// TIA Portal V17 export
// export: Created 2025-06-26T06:33:59.0377873Z, ExportSetting WithDefaults, DisplayName Totally Integrated Automation Portal, DisplayVersion V17 Update 8, DisplayName TIA Portal Openness, DisplayVersion V17 Update 8, DisplayName TIA Portal Version Control Interface, DisplayVersion V17, DisplayName STEP 7 Professional, DisplayVersion V17 Update 8, DisplayName STEP 7 Safety, DisplayVersion V17 Update 6, DisplayName WinCC Advanced, DisplayVersion V17 Update 8
DATA_BLOCK "DB_Heatbooster"   // DB19
{ S7_Optimized_Access := 'TRUE' }
VERSION : 0.1
// stored: AutoNumber true, DBAccessibleFromOPCUA true, IsOnlyStoredInLoadMemory false, IsRetainMemResEnabled false, IsWriteProtectedInAS false, MemoryReserve 0
   VAR
      AI : Struct
         HBL_TT_502 { S7_SetPoint := 'True'} : "stCalcValue";   // Compressor discharge popoff temperature
         HBL_PT_503 { S7_SetPoint := 'True'} : "stCalcValue";   // Compressor discharge pressure
         HBL_TT_504 { S7_SetPoint := 'True'} : "stCalcValue";   // Compressor discharge temperature
         HBL_LT_510 { S7_SetPoint := 'True'} : "stCalcValue";   // Steam generator condensate level
         HBL_PT_511 { S7_SetPoint := 'True'} : "stCalcValue";   // Heat sink discharge pressure
         HBL_TT_512 { S7_SetPoint := 'True'} : "stCalcValue";   // Heat sink discharge temperature
         HBL_TT_516 { S7_SetPoint := 'True'} : "stCalcValue";   // Steam generator suction temperature
         HBL_PT_517 { S7_SetPoint := 'True'} : "stCalcValue";   // Steam generator suction pressure
         HBL_TT_518 { S7_SetPoint := 'True'} : "stCalcValue";   // Heat sink discharge process temperature
         HBL_PT_519 { S7_SetPoint := 'True'} : "stCalcValue";   // Heat sink discharge process pressure
         HBL_FT_520 { S7_SetPoint := 'True'} : "stCalcValue";   // Refrigerant flow
         HBL_TT_530 { S7_SetPoint := 'True'} : "stCalcValue";   // Expansion valve B discharge temperature
         HBL_PT_531 { S7_SetPoint := 'True'} : "stCalcValue";   // Expansion valve B discharge pressure
         HBL_TT_532 { S7_SetPoint := 'True'} : "stCalcValue";   // Heat source discharge B temperature
         HBL_TT_533 { S7_SetPoint := 'True'} : "stCalcValue";   // Evaporator B discharge temperature
         HBL_PT_534 { S7_SetPoint := 'True'} : "stCalcValue";   // Evaporator B discharge pressure
         HBL_AT_535 { S7_SetPoint := 'True'} : "stCalcValue";   // Evaporator B steam quality
         HBL_TT_540 { S7_SetPoint := 'True'} : "stCalcValue";   // Expansion valve A discharge temperature
         HBL_PT_541 { S7_SetPoint := 'True'} : "stCalcValue";   // Expansion valve A discharge pressure
         HBL_TT_542 { S7_SetPoint := 'True'} : "stCalcValue";   // Heat source discharge temperature
         HBL_TT_543 { S7_SetPoint := 'True'} : "stCalcValue";   // Evaporator A discharge temperature
         HBL_PT_544 { S7_SetPoint := 'True'} : "stCalcValue";   // Evaporator A discharge pressure
         HBL_AT_545 { S7_SetPoint := 'True'} : "stCalcValue";   // Evaporator A steam quality
         HBL_TT_546 { S7_SetPoint := 'True'} : "stCalcValue";   // Heat source suction temperature
         HBL_PT_547 { S7_SetPoint := 'True'} : "stCalcValue";   // Heast source suction pressure
         HBL_TT_571 { S7_SetPoint := 'True'} : "stCalcValue";   // Compressor suction temperature
         HBL_PT_572 { S7_SetPoint := 'True'} : "stCalcValue";   // Compressor suction pressure
         HBL_TT_573 { S7_SetPoint := 'True'} : "stCalcValue";   // Expansion valve suction temperature
         HBL_LT_610 { S7_SetPoint := 'True'} : "stCalcValue";   // HP receiver refrigerant level
         HBL_TT_611 { S7_SetPoint := 'True'} : "stCalcValue";   // Steam generator discharge temperature
         HBL_PT_612 { S7_SetPoint := 'True'} : "stCalcValue";   // Steam generator discharge pressure
         HBL_CT_615 { S7_SetPoint := 'True'} : "stCalcValue";   // Gas detector PSV discharge pipe
         HBL_PT_618 { S7_SetPoint := 'True'} : "stCalcValue";   // HP Receiver pressure
         HBL_PT_635 { S7_SetPoint := 'True'} : "stCalcValue";   // Oil separator stage 1 oil return pressure
         HBL_PT_636 { S7_SetPoint := 'True'} : "stCalcValue";   // Oil separator stage 2 oil return pressure
         HBL_LT_650 { S7_SetPoint := 'True'} : "stCalcValue";   // Heat source condensate buffer tank level
         HBL_PT_651 { S7_SetPoint := 'True'} : "stCalcValue";   // Heat source condensate buffer tank pressure
         HBL_PT_701 { S7_SetPoint := 'True'} : "stCalcValue";   // Filter dryer suction pressure
         HBL_PT_702 { S7_SetPoint := 'True'} : "stCalcValue";   // Filter dryer discharge pressure
         HBL_PT_703 { S7_SetPoint := 'True'} : "stCalcValue";   // Filter dryer differential pressure
         CPC_LT_870 { S7_SetPoint := 'True'} : "stCalcValue";   // CPC tank refrigerant level
         CPC_TT_871 { S7_SetPoint := 'True'} : "stCalcValue";   // CPC tank refrigerant temperature
         CPC_PT_872 { S7_SetPoint := 'True'} : "stCalcValue";   // CPC tank refrigerant pressure
         CPC_PT_862 { S7_SetPoint := 'True'} : "stCalcValue";   // CPC pump discharge pressure
         HBL_TT_901 { S7_SetPoint := 'True'} : "stCalcValue";   // Heat sink suction temperature
         HBL_PT_902 { S7_SetPoint := 'True'} : "stCalcValue";   // Heat sink suction pressure
         HBL_TT_03 { S7_SetPoint := 'True'} : "stCalcValue";   // Oil sump oil temperature
         HBL_TT_16 { S7_SetPoint := 'True'} : "stCalcValue";   // Container air temperature
         HBL_TT_17 { S7_SetPoint := 'True'} : "stCalcValue";   // Control cabinet air temperature
         HBL_TT_18 { S7_SetPoint := 'True'} : "stCalcValue";   // Ambient air temperature
         HBL_TT_20 { S7_SetPoint := 'True'} : "stCalcValue";   // Compressor motor winding temperature
         HBL_TT_21 { S7_SetPoint := 'True'} : "stCalcValue";   // Oil sump wall temperature left
         HBL_TT_22 { S7_SetPoint := 'True'} : "stCalcValue";   // Oil sump wall temperature right
         HBL_TT_23 { S7_SetPoint := 'True'} : "stCalcValue";   // Compressor motor U-winding temperature
         HBL_TT_24 { S7_SetPoint := 'True'} : "stCalcValue";   // Compressor motor V-winding temperature
         HBL_TT_25 { S7_SetPoint := 'True'} : "stCalcValue";   // Compressor motor W-winding temperature
         HBL_TT_26 { S7_SetPoint := 'True'} : "stCalcValue";   // Compressor motor D bearing temperature
         HBL_TT_27 { S7_SetPoint := 'True'} : "stCalcValue";   // Compressor motor N bearing temperature
         HBL_PT_05 { S7_SetPoint := 'True'} : "stCalcValue";   // Crankcase gas pressure
         HBL_PT_06 { S7_SetPoint := 'True'} : "stCalcValue";   // Oil pump discharge pressure
         HBL_PT_17 { S7_SetPoint := 'True'} : "stCalcValue";   // Oil gallery pressure
         HBL_CT_01 { S7_SetPoint := 'True'} : "stCalcValue";   // Gas detector Heatbooster (optional)
         HBL_CT_03 { S7_SetPoint := 'True'} : "stCalcValue";   // Gas detector container (optional)
         SSC_TT_01 { S7_SetPoint := 'True'} : "stCalcValue";   // SSC seal suction temperature
         SSC_TT_02 { S7_SetPoint := 'True'} : "stCalcValue";   // SSC seal discharge temperature
         SSC_TT_03 { S7_SetPoint := 'True'} : "stCalcValue";   // SSC barrier fluid circulation pump suction temperature
         SSC_TT_04 { S7_SetPoint := 'True'} : "stCalcValue";   // SSC barrier fluid heat exchanger temperature
         SSC_PIT_01 { S7_SetPoint := 'True'} : "stCalcValue";   // SSC barrier fluid accumulator pressure
         SSC_PDT_01 { S7_SetPoint := 'True'} : "stCalcValue";   // SSC barrier fluid circulation pump differential pressure
         SSC_LT_01 { S7_SetPoint := 'True'} : "stCalcValue";   // SSC barrier fluid reservoir level
         HBL_VT_01 { S7_SetPoint := 'True'} : "stCalcValue";   // [?] Oil sump oil viscosity
         HBL_TT_36 { S7_SetPoint := 'True'} : "stCalcValue";   // [C] Oil sump oil viscosity probe temperature
      END_STRUCT;
      Calc : Struct
         Compressor : Struct
            CrankcaseSaturationTemperature { S7_SetPoint := 'True'} : "stCalcValue";   // C
            CrankcaseSuperheat { S7_SetPoint := 'True'} : "stCalcValue";   // C
            VolumetricEfficiency { S7_SetPoint := 'True'} : "stCalcValue";   // %
            IsentropicEfficiency { S7_SetPoint := 'True'} : "stCalcValue";   // %
            Massflow { S7_SetPoint := 'True'} : "stCalcValue";   // kg/h
         END_STRUCT;
         HeatSink : Struct
            DeltaT { S7_SetPoint := 'True'} : "stCalcValue";
            Pinch { S7_SetPoint := 'True'} : "stCalcValue";
            HeatRate { S7_SetPoint := 'True'} : "stCalcValue";
            DeltaP { S7_SetPoint := 'True'} : "stCalcValue";
            Massflow { S7_SetPoint := 'True'} : "stCalcValue";
         END_STRUCT;
         HeatSource : Struct
            DeltaT { S7_SetPoint := 'True'} : "stCalcValue";
            Pinch { S7_SetPoint := 'True'} : "stCalcValue";
            HeatRate { S7_SetPoint := 'True'} : "stCalcValue";
            DeltaP { S7_SetPoint := 'True'} : "stCalcValue";
            TemperatureRateOfChange { S7_SetPoint := 'True'} : "stCalcValue";
            Massflow { S7_SetPoint := 'True'} : "stCalcValue";
         END_STRUCT;
         HighPressPart : Struct
            CompressorSaturationTemperature { S7_SetPoint := 'True'} : "stCalcValue";
            CompressorSuperheat { S7_SetPoint := 'True'} : "stCalcValue";
            CondenserSaturationTemperature { S7_SetPoint := 'True'} : "stCalcValue";
            CondenserSubcooling { S7_SetPoint := 'True'} : "stCalcValue";
            ExpansionValveSubcooling { S7_SetPoint := 'True'} : "stCalcValue";
            CondenserDeltaP { S7_SetPoint := 'True'} : "stCalcValue";
         END_STRUCT;
         LowPressPart : Struct
            EvaporatorSuperheat { S7_SetPoint := 'True'} : "stCalcValue";
            CompressorSuperheat { S7_SetPoint := 'True'} : "stCalcValue";
            EvaporatorSaturationTemperature { S7_SetPoint := 'True'} : "stCalcValue";
            CompressorSaturationTemperature { S7_SetPoint := 'True'} : "stCalcValue";
         END_STRUCT;
         System : Struct
            Quality { S7_SetPoint := 'True'} : "stCalcValue";
            COP { S7_SetPoint := 'True'} : "stCalcValue";
            ElectricalPower { S7_SetPoint := 'True'} : "stCalcValue";
            TemperatureLift { S7_SetPoint := 'True'} : "stCalcValue";
            MotorEfficiency { S7_SetPoint := 'True'} : "stCalcValue";
            FMEP { S7_SetPoint := 'True'} : "stCalcValue";
         END_STRUCT;
         Auxiliary : Struct
            ShaftSealDeltaT { S7_SetPoint := 'True'} : "stCalcValue";
            CPCPumpDeltaP { S7_SetPoint := 'True'} : "stCalcValue";
         END_STRUCT;
         Misc : Struct
            EvaporatorDischargePressureMean { S7_SetPoint := 'True'} : "stCalcValue";
            EvaporatorDischargeTemperatureMin { S7_SetPoint := 'True'} : "stCalcValue";
            EvaporatorDischargeTemperatureMean { S7_SetPoint := 'True'} : "stCalcValue";
            OilFilterDeltaP { S7_SetPoint := 'True'} : "stCalcValue";
         END_STRUCT;
      END_STRUCT;
      DI : Struct
         HBL_FS_01 : Bool;
         HBL_FS_02 : Bool;
         HBL_LS_632 : Bool;
         HBL_LS_633 : Bool;
         CPC_LS_864 : Bool;
         VPNUserConnected : Bool;
      END_STRUCT;
      "DO" : Struct
         HBL_EC_01 : Bool;
         HBL_EC_02 : Bool;
         HBL_HV_630 : Bool;
         HBL_HV_114 : Bool;
         HBL_HV_115 : Bool;
         HBL_HV_860 : Bool;
         HBL_HV_861 : Bool;
         SSC_P_01 : Bool;
         SSC_F_01 : Bool;
         SSC_P_02 : Bool;
         CPC_P_01 : Bool;
         SpareContactor1 : Bool;
         SpareContactor2 : Bool;
         HBL_HV_631 : Bool;
      END_STRUCT;
      Inverter : Struct
         HBL_SC_01_A1 { S7_SetPoint := 'True'} : "stCalcValue";   // Container ventilation fan speed
         HBL_SC_01_A2 { S7_SetPoint := 'True'} : "stCalcValue";   // Container ventilation fan torque
         HBL_SC_01_A3 { S7_SetPoint := 'True'} : "stCalcValue";   // Container ventilation fan power
         HBL_SC_02_A1 { S7_SetPoint := 'True'} : "stCalcValue";   // Compressor lubrication pump speed
         HBL_SC_02_A2 { S7_SetPoint := 'True'} : "stCalcValue";   // Compressor lubrication pump torque
         HBL_SC_02_A3 { S7_SetPoint := 'True'} : "stCalcValue";   // Compressor lubrication pump power
         HBL_SC_03_A1 { S7_SetPoint := 'True'} : "stCalcValue";   // CPC pump speed
         HBL_SC_03_A2 { S7_SetPoint := 'True'} : "stCalcValue";   // CPC pump torque
         HBL_SC_03_A3 { S7_SetPoint := 'True'} : "stCalcValue";   // CPC pump power
         HBL_SC_10_A1 { S7_SetPoint := 'True'} : "stCalcValue";   // Compressor motor speed
         HBL_SC_10_A2 { S7_SetPoint := 'True'} : "stCalcValue";   // Compressor motor torque
         HBL_SC_10_A3 { S7_SetPoint := 'True'} : "stCalcValue";   // Compressor motor power
      END_STRUCT;
      Valve : Struct
         HBL_HCV_576_A1 : "stCalcValue";   // Expansion Valve A
         HBL_HCV_578_A1 : "stCalcValue";   // Expansion Valve B
         HBL_HCV_577_A1 { S7_SetPoint := 'True'} : "stCalcValue";   // Expansion Valve A2
         HBL_HCV_579_A1 { S7_SetPoint := 'True'} : "stCalcValue";   // Expansion Valve B2
         HBL_HCV_515_A1 { S7_SetPoint := 'True'} : "stCalcValue";   // Heat sink condensate blowdown flow control valve
         HBL_HCV_575_A1 { S7_SetPoint := 'True'} : "stCalcValue";   // Recuperator oil drain valve
         HBL_HCV_616_A1 { S7_SetPoint := 'True'} : "stCalcValue";   // Recuperator bypass valve
         HBL_HCV_700_A1 { S7_SetPoint := 'True'} : "stCalcValue";   // Oil recovery refrigerant blowdown valve
         HBL_HCV_514_A1 { S7_SetPoint := 'True'} : "stCalcValue";   // Heat sink discharge pressure control valve
         HBL_HCV_548_A1 { S7_SetPoint := 'True'} : "stCalcValue";   // Heat source suction pressure control valve
      END_STRUCT;
   END_VAR
BEGIN
END_DATA_BLOCK
